vlevo abs 6 / Posición final izq abs 6 / Position finale gauche abs 6 / véghelyzet balra abs 6 / Pos finale a sx ass. 6 / Poł. krańc. lewej abs 6 / Конечное положение влево абс. 6 / Ändläge vänster abs 6 / Posição final esq abs 6 / Poziţie de capăt stânga abs 6 / End position left abs 6'; 626 'Bew aktiv rechts sym / Movement active right sym / 右侧运动生效系统 6 / Pohyb akt vpravo sym 6 / Mov act dcha simb 6 / Dépl act droite sym 6 / mozgás aktív jobbra sym 6 / Mov att a dx simm. 6 / Ruch aktyw. lewo sym 6 / Движение активно вправо симв. 6 / Rörelse aktiv höger sym 6 / Movmt atv dir sym 6 / Depl. activă dreapta sim 6 / Movmt act right sym 6'; 627 'Bew aktiv rechts abs / Movement active right abs / 右侧运动生效绝对 6 / Pohyb akt vpravo abs 6 / Mov act dcha abs 6 / Dépl act droite abs 6 / mozgás aktív jobbra abs 6 / Mov att a dx ass. 6 / Ruch aktyw. prawo 6 / Движение активно вправо абс. 6 / Rörelse aktiv höger abs 6 / Movmt atv direito abs 6 / Depl. activă dreapta abs 6 / Movmt act right abs 6'; 628 'Endlage rechts sym / End position right sym / 右侧最终位置系统 6 / Koncová poloha vpravo sym 6 / Posición final dcha simb 6 / Position finale droite sym 6 / véghelyzet jobbra sym 6 / Pos finale a dx simm. 6 / Poł. krańc. prawej sym 6 / Конечное положение вправо симв. 6 / Ändläge höger sym 6 / Posição final dir sym 6 / Poziţie de capăt dreapta sim 6 / End position right sym 6'; 629 'Endlage rechts abs / End position right abs / 右侧最终位置绝对 6 / Koncová poloha vpravo abs 6 / Posición final derecha abs 6 / Position finale droite abs 6 / véghelyzet jobbra absz 6 / Pos finale a dx ass. 6 / Położenie krańcowe prawe abs 6 / Конечное положение вправо abs 6 / Ändläge höger abs 6 / Posição final direita abs 6 / Poziţie de capăt dreapta abs 6 / End position right abs 6'; 630 'Funktion sym / Function sym / 功能系统 6 / Funkce sym 6 / Función simb 6 / Fonction sym 6 / sym 6 funkció / Funzione simm. 6 / Funkcja sym 6 / Функция симв. 6 / Funktion sym 6 / Função sym 6 / Funcţie sim 6 / Function sym 6'; 631 'Funktion abs / Function abs / 功能绝对 6 / Funkce abs 6 / Función abs 6 / Fonction abs 6 / abs 6 funkció / Funzione ass. 6 / Funkcja abs 6 / Функция абс. 6 / Funktion abs 6 / Função abs 6 / Funcţie abs 6 / Function abs 6'; 632 'Bew aktiv links sym / Movement active left sym / 左侧运动生效系统 6 / Pohyb akt vlevo sym 6 / Mov act izq simb 6 / Dépl act gauche sym 6 / mozgás aktív balra sym 6 / Mov att a sx simm. 6 / Ruch aktyw. lewo sym 6 / Движение активно влево симв. 6 / Rörelse aktiv vänster sym 6 / Movmt atv esq sym 6 / Depl. activă stânga sim 6 / Movmt act left sym 6'; 633 'Bew aktiv links abs / Movement active left abs / 左侧运动生效绝对 6 / Pohyb akt vlevo abs 6 / Mov act izq abs 6 / Dépl act gauche abs 6 / mozgás aktív balra abs 6 / Mov att a sx ass. 6 / Ruch aktyw. lewo abs 6 / Движение активно влево абс. 6 / Rörelse aktiv vänster abs 6 / Movmt atv esq abs 6 / Depl. activă stânga abs 6 / Movmt act left abs 6'; 634 'Endlage links sym / End position left sym / 左侧最终位置系统 6 / Koncová poloha vlevo sym 6 / Posición final izq simb 6 / Position finale gauche sym 6 / véghelyzet balra sym 6 / Pos finale a sx simm. 6 / Poł. krańc. lewej sym 6 / Конечное положение влево сим. 6 / Ändläge vänster sym 6 / Posição final esq sym 6 / Poziţie de capăt stânga sim 6 / End position left sym 6'; 635 'Endlage links abs / End position left abs / 左侧最终位置绝对 6 / Koncová poloha vlevo abs 6 / Posición final izq abs 6 / Position finale gauche abs 6 / véghelyzet balra abs 6 / Pos finale a sx ass. 6 / Poł. krańc. lewej abs 6 / Конечное положение влево абс. 6 / Ändläge vänster abs 6 / Posição final esq abs 6 / Poziţie de capăt stânga abs 6 / End position left abs 6'; 636 'Bew aktiv rechts sym / Movement active right sym / 右侧运动生效系统 6 / Pohyb akt vpravo sym 6 / Mov act dcha simb 6 / Dépl act droite sym 6 / mozgás aktív jobbra sym 6 / Mov att a dx simm. 6 / Ruch aktyw. lewo sym 6 / Движение активно вправо симв. 6 / Rörelse aktiv höger sym 6 / Movmt atv dir sym 6 / Depl. activă dreapta sim 6 / Movmt act right sym 6'; 637 'Bew aktiv rechts abs / Movement active right abs / 右侧运动生效绝对 6 / Pohyb akt vpravo abs 6 / Mov act dcha abs 6 / Dépl act droite abs 6 / mozgás aktív jobbra abs 6 / Mov att a dx ass. 6 / Ruch aktyw. prawo 6 / Движение активно вправо абс. 6 / Rörelse aktiv höger abs 6 / Movmt atv direito abs 6 / Depl. activă dreapta abs 6 / Movmt act right abs 6'; 638 'Endlage rechts sym / End position right sym / 右侧最终位置系统 6 / Koncová poloha vpravo sym 6 / Posición final dcha simb 6 / Position finale droite sym 6 / véghelyzet jobbra sym 6 / Pos finale a dx simm. 6 / Poł. krańc. prawej sym 6 / Конечное положение вправо симв. 6 / Ändläge höger sym 6 / Posição final dir sym 6 / Poziţie de capăt dreapta sim 6 / End position right sym 6'; 639 'Endlage rechts abs / End position right abs / 右侧最终位置绝对 6 / Koncová poloha vpravo abs 6 / Posición final derecha abs 6 / Position finale droite abs 6 / véghelyzet jobbra absz 6 / Pos finale a dx ass. 6 / Położenie krańcowe prawe abs 6 / Конечное положение вправо abs 6 / Ändläge höger abs 6 / Posição final direita abs 6 / Poziţie de capăt dreapta abs 6 / End position right abs 6'

text list "Overview": 1 'FG 1'; 2 'FG 2'; 3 'FG 3'; 4 'FG 4'; 5 'FG 5'; 10 'FG Transport'; 0 'FG x'

text list "Header_Line_2": 0 ''; 1 ''

text list "StationState": 0 'Bearbeitung / Processing'; 1 'Störung / Fault'; 2 'Nicht benötigt / Not required'; 3 'Nicht in Produktion / Not in production'; 4 'Wartet auf Bediener / Waiting for operator'; 5 'Ausgabe blockiert / Output blocked'; 6 'Wartet auf Eingabe / Waiting for infeed'

Template "Vorlage_1" 800x420
   Button "Beenden" at 720,360 size 78x58; TextOff 'Beenden / Exit'; PictureOff "ExitRuntime_TP700_Comfort_TR"; PictureOn "ExitRuntime_TP700_Comfort_TR"
      on Release: StopRuntime(0)
   Button "Template_Button" at 640,360 size 78x58; TextOff 'Meldungen / Messages'; PictureOff "meldungen_48"
      on Click: function_ef3f5d25("Meldefenster_Anstehend", -1)
   Button "Template_Button_1" at 560,360 size 78x58; TextOff 'Text'
   Button "Template_Button_2" at 480,360 size 78x58; TextOff 'Text'
   Button "Template_Button_3" at 400,360 size 78x58; TextOff 'Text'
   Button "Template_Button_4" at 321,360 size 78x58; TextOff 'Text'
   Button "Template_Button_5" at 241,360 size 78x58; TextOff 'Taktzeiten / Cycle times'; PictureOff "taktzeiten_48"
      on Release: ActivateScreen("101_Taktzeiten", 0)
   Button "Template_Button_6" at 161,360 size 78x58; TextOff 'Übersicht / Overview'; PictureOff "uebersicht_48"
      on Release: ActivateScreen("2_Übersicht", 0)
   Button "Template_Button_7" at 81,360 size 78x58; TextOff 'zurück / back'; PictureOff "zurueck_48"
      on Click: function_efd93a16()
   Button "Startbild" at 1,360 size 78x58; TextOff 'Startbild / Start screen'; PictureOff "NavigateHome_TP700_Comfort_TR"; PictureOn "NavigateHome_TP700_Comfort_TR"
      on Release: ActivateScreen("1_Grundbild", 0)
   AlarmView "Meldeanzeige_Nichtquittiert" at 0,0 size 800x20

screen "1_Grundbild" 800x420, template "Vorlage_1"
   on GenerateScreen: SetTag("Header_Line_1", 1)
   Button "HmiScreenItemData" at 36,60 size 159x47; TextOff 'Automatik / Automatic'; PictureOff "Navigates to Automatik for TP700 Comfort 17.0.0.0"; PictureOn "Navigates to Automatik for TP700 Comfort 17.0.0.0"
      on Release: ActivateScreen("100_Automatik", 0)
   Button "HmiScreenItemData_1" at 36,119 size 159x47; TextOff 'Einrichten / Setup'; PictureOff "Navigates to Einrichten for TP700 Comfort 17.0.0.0"; PictureOn "Navigates to Einrichten for TP700 Comfort 17.0.0.0"
      on Release: ActivateScreen("10_Einrichten", 0)
   Button "HmiScreenItemData_3" at 36,178 size 159x47; TextOff 'Systembilder / System screens'; PictureOff "Navigates to Systembilder for TP700 Comfort 17.0.0.0"; PictureOn "Navigates to Systembilder for TP700 Comfort 17.0.0.0"
      on Release: ActivateScreen("1000_Systembilder", 0)

screen "100_Automatik" 800x420, template "Vorlage_1"
   on GenerateScreen: SetTag("Header_Line_1", 100)
   TextField "Textfeld_1" at 11,34 size 365x42; Text 'Maschine leerfahren / Empty machine'
   Switch "Schalter_1" at 376,34 size 83x42; CaptionText 'Umschalten'; TextOff 'Aus / Off'; TextOn 'Ein / On'
      ProcessValue <- "MachineGlobals_emptying"
      Appearance <- "MachineGlobals_emptying"
   TextField "Textfeld_2" at 11,76 size 365x42; Text 'FG05 leerfahren / Empty FG05'
   Switch "Schalter_2" at 376,76 size 83x42; CaptionText 'Umschalten'; TextOff 'Aus / Off'; TextOn 'Ein / On'
      ProcessValue <- "FG05Globals_emptying"
      Appearance <- "FG05Globals_emptying"
   TextField "Textfeld_3" at 11,118 size 365x42; Text 'FG01 Laser einschalten / FG01 Switch on laser'
   Switch "Schalter_3" at 376,118 size 83x42; CaptionText 'Umschalten'; TextOff 'Aus / Off'; TextOn 'Ein / On'
      ProcessValue <- "FG01Globals_laserOn"
      Appearance <- "FG01Globals_laserOn"

screen "10_Einrichten" 800x420, template "Vorlage_1"
   on GenerateScreen: SetTag("Header_Line_1", 10)
   Button "HmiScreenItemData_1" at 35,41 size 159x47; TextOff 'FG 1 / Einrichtfunktionen'; TextOn 'Einrichtfunktionen'; PictureOff "Navigates to Einrichtfunktionen for TP700 Comfort 17.0.0.0"; PictureOn "Navigates to Einrichtfunktionen for TP700 Comfort 17.0.0.0"
      on Release: ActivateScreen("12_Einrichtfunktionen", 0); SetTag("HmiManualMovement_selection_station", 1)
      Visibility <- "xExists"
   Button "HmiScreenItemData_2" at 35,100 size 159x47; TextOff 'FG 2 / Einrichtfunktionen'; TextOn 'Einrichtfunktionen'; PictureOff "Navigates to Einrichtfunktionen for TP700 Comfort 17.0.0.0"; PictureOn "Navigates to Einrichtfunktionen for TP700 Comfort 17.0.0.0"
      on Release: ActivateScreen("12_Einrichtfunktionen", 0); SetTag("HmiManualMovement_selection_station", 2)
      Visibility <- "xExists"
   Button "HmiScreenItemData_3" at 35,160 size 159x47; TextOff 'FG 3 / Einrichtfunktionen'; TextOn 'Einrichtfunktionen'; PictureOff "Navigates to Einrichtfunktionen for TP700 Comfort 17.0.0.0"; PictureOn "Navigates to Einrichtfunktionen for TP700 Comfort 17.0.0.0"
      on Release: ActivateScreen("12_Einrichtfunktionen", 0); SetTag("HmiManualMovement_selection_station", 3)
      Visibility <- "xExists"
   Button "HmiScreenItemData_4" at 35,223 size 159x47; TextOff 'FG 4 / Einrichtfunktionen'; TextOn 'Einrichtfunktionen'; PictureOff "Navigates to Einrichtfunktionen for TP700 Comfort 17.0.0.0"; PictureOn "Navigates to Einrichtfunktionen for TP700 Comfort 17.0.0.0"
      on Release: ActivateScreen("12_Einrichtfunktionen", 0); SetTag("HmiManualMovement_selection_station", 4)
      Visibility <- "xExists"
   Button "HmiScreenItemData_5" at 35,282 size 159x47; TextOff 'FG 5 / Einrichtfunktionen'; TextOn 'Einrichtfunktionen'; PictureOff "Navigates to Einrichtfunktionen for TP700 Comfort 17.0.0.0"; PictureOn "Navigates to Einrichtfunktionen for TP700 Comfort 17.0.0.0"
      on Release: ActivateScreen("12_Einrichtfunktionen", 0); SetTag("HmiManualMovement_selection_station", 5)
      Visibility <- "xExists"
   Button "HmiScreenItemData_6" at 232,282 size 159x47; TextOff 'FG Transport / Einrichtfunktionen'; TextOn 'Einrichtfunktionen'; PictureOff "Navigates to Einrichtfunktionen for TP700 Comfort 17.0.0.0"; PictureOn "Navigates to Einrichtfunktionen for TP700 Comfort 17.0.0.0"
      on Release: ActivateScreen("12_Einrichtfunktionen", 0); SetTag("HmiManualMovement_selection_station", 10)
      Visibility <- "xExists"
   Button "HmiScreenItemData_7" at 232,41 size 159x47; TextOff 'FG 6 / Einrichtfunktionen'; TextOn 'Einrichtfunktionen'; PictureOff "Navigates to Einrichtfunktionen for TP700 Comfort 17.0.0.0"; PictureOn "Navigates to Einrichtfunktionen for TP700 Comfort 17.0.0.0"
      on Release: ActivateScreen("12_Einrichtfunktionen", 0); SetTag("HmiManualMovement_selection_station", 1)
      Visibility <- "xExists"
   Button "HmiScreenItemData_8" at 232,100 size 159x47; TextOff 'FG 7 / Einrichtfunktionen'; TextOn 'Einrichtfunktionen'; PictureOff "Navigates to Einrichtfunktionen for TP700 Comfort 17.0.0.0"; PictureOn "Navigates to Einrichtfunktionen for TP700 Comfort 17.0.0.0"
      on Release: ActivateScreen("12_Einrichtfunktionen", 0); SetTag("HmiManualMovement_selection_station", 1)
      Visibility <- "xExists"
   Button "HmiScreenItemData_9" at 232,159 size 159x47; TextOff 'FG 8 / Einrichtfunktionen'; TextOn 'Einrichtfunktionen'; PictureOff "Navigates to Einrichtfunktionen for TP700 Comfort 17.0.0.0"; PictureOn "Navigates to Einrichtfunktionen for TP700 Comfort 17.0.0.0"
      on Release: ActivateScreen("12_Einrichtfunktionen", 0); SetTag("HmiManualMovement_selection_station", 1)
      Visibility <- "xExists"
   Button "HmiScreenItemData_10" at 232,218 size 159x47; TextOff 'FG 9 / Einrichtfunktionen'; TextOn 'Einrichtfunktionen'; PictureOff "Navigates to Einrichtfunktionen for TP700 Comfort 17.0.0.0"; PictureOn "Navigates to Einrichtfunktionen for TP700 Comfort 17.0.0.0"
      on Release: ActivateScreen("12_Einrichtfunktionen", 0); SetTag("HmiManualMovement_selection_station", 1)
      Visibility <- "xExists"

screen "12_Einrichtfunktionen" 800x420, template "Vorlage_1"
   on GenerateScreen: SetTag("Header_Line_1", 12); SetTag("Header_Line_2", 1)
   on ClearScreen: SetTag("HmiManualMovement_selection_station", 0); SetTag("Header_Line_2", 0)
   Rectangle "recExecuteLeft1" at 0,22 size 285x72
      Visibility <- "showRecLeft"
   Rectangle "recRuntime1" at 287,22 size 226x72
      Visibility <- "showName"
   Rectangle "recExecuteRight1" at 515,22 size 285x72
      Visibility <- "showRecRight"
   Rectangle "recConfirmExecuteLeft1" at 60,26 size 29x29
      Appearance <- "workAct"
      Visibility <- "isExecutableLeft"
   Rectangle "recFinalPositionLeft1" at 60,61 size 29x29
      Appearance <- "inWorkPos"
      Visibility <- "hasEndPositionLeft"
   Polygon "polExecutabilityLeft1" at 2,30 size 51x55
      Appearance <- "workIsInterlocked"
      Visibility <- "isExecutableLeft"
   SymbolicIOField "seaConfirmExecuteLeft1" at 92,26 size 193x29; TextOn '1'; TextOff '0'; TextList "Setup"
      ProcessValue <- "textlistFunctionExecuteLeft"
      Visibility <- "isExecutableLeft"
   SymbolicIOField "seaFinalPositionLeft1" at 92,61 size 193x29; TextOn '1'; TextOff '0'; TextList "Setup"
      ProcessValue <- "textlistFunctionFinalPosLeft"
      Visibility <- "hasEndPositionLeft"
   Rectangle "recFinalPositionRight1" at 711,61 size 29x29
      Appearance <- "inHomePos"
      Visibility <- "hasEndPositionRight"
   Polygon "polExecutabilityRight1" at 747,30 size 51x55
      Appearance <- "homeIsInterlocked"
      Visibility <- "isExecutableRight"
   SymbolicIOField "seaFunction1" at 287,26 size 226x29; TextOn '1'; TextOff '0'; TextList "Setup"
      ProcessValue <- "textlistFunctionName"
      Visibility <- "showName"
   SymbolicIOField "seaConfirmExecuteRight1" at 515,26 size 193x29; TextOn '1'; TextOff '0'; TextList "Setup"
      ProcessValue <- "textlistFunctionExecuteRight"
      Visibility <- "isExecutableRight"
   SymbolicIOField "seaFinalPositionRight1" at 515,61 size 193x29; TextOn '1'; TextOff '0'; TextList "Setup"
      ProcessValue <- "textlistFunctionFinalPosRight"
      Visibility <- "hasEndPositionRight"
   IOField "eaPosition1" at 287,61 size 226x29; FormatPattern s999999999.999
      ProcessValue <- "value"
      Visibility <- "showValue"
   Rectangle "recConfirmExecuteRight1" at 711,26 size 29x29
      Appearance <- "homeAct"
      Visibility <- "isExecutableRight"
   Button "btnRight1" at 515,22 size 285x72; TextOn 'Texto / Texte / Testo / 文本 / Text / Szöv / Текст / Tekst'; TextOff 'Texto / Texte / Testo / 文本 / Text / Szöv / Текст / Tekst'
      on Release: SetTag("moveHomePos", 0)
      on Press: SetTag("moveHomePos", 1)
      ObjectEnable <- "isExecutableRight"
   Button "btnLeft1" at 0,22 size 285x72; TextOn 'Texto / Texte / Testo / 文本 / Text / Szöv / Текст / Tekst'; TextOff 'Texto / Texte / Testo / 文本 / Text / Szöv / Текст / Tekst'
      on Release: SetTag("moveWorkPos", 0)
      on Press: SetTag("moveWorkPos", 1)
      ObjectEnable <- "isExecutableLeft"
   TextField "txtPage" at 524,326 size 120x29; Text 'Seite / Página / Page / Pagina / 页 / Stránka / Oldal / Страница / stron / Sida / Pagină'
   IOField "eaActualPage" at 654,326 size 41x29; FormatPattern 999
      ProcessValue <- "HmiManualMovement_selection_page"
   TextField "txtOf" at 696,326 size 56x29; Text 'von / de / di / 之 / of / od / tól / из / z / av / din'
   IOField "eaNumberOfPages" at 753,326 size 41x29; FormatPattern 999
      ProcessValue <- "HmiManualMovement_selection_ofMaxPages"
   Group "Function 1" at 0,22 size 800x72; TextList "Setup"
   Group "Function 2" at 0,96 size 800x72; TextList "Setup"
   Group "Function 3" at 0,170 size 800x72; TextList "Setup"
   Group "Function 4" at 0,244 size 800x72; TextList "Setup"
   Button "Template_Button" at 640,360 size 78x58; TextOff 'Seite + Page +'; PictureOff "seite_vor_48"
      on Press: SetBit("HmiManualMovement_selection_nextPage")
   Button "Template_Button_1" at 560,360 size 78x58; TextOff 'Seite - Page -'; PictureOff "seite_zurueck_48"
      on Press: SetBit("HmiManualMovement_selection_previousPage")
   Button "Template_Button_2" at 480,360 size 78x58; TextOff 'Symbol Absolut Symbolic Absolute'; PictureOff "symbol_absolut_48"
      on Press: InvertBit("HmiManualMovement_selection_showSymbols")
   Rectangle "recExecuteLeft1_1" at 0,96 size 285x72
      Visibility <- "showRecLeft"
   Rectangle "recRuntime1_1" at 287,96 size 226x72
      Visibility <- "showName"
   Rectangle "recExecuteRight1_1" at 515,96 size 285x72
      Visibility <- "showRecRight"
   Rectangle "recConfirmExecuteLeft1_1" at 60,100 size 29x29
      Appearance <- "workAct"
      Visibility <- "isExecutableLeft"
   Rectangle "recFinalPositionLeft1_1" at 60,135 size 29x29
      Appearance <- "inWorkPos"
      Visibility <- "hasEndPositionLeft"
   Polygon "polExecutabilityLeft1_1" at 2,104 size 51x55
      Appearance <- "workIsInterlocked"
      Visibility <- "isExecutableLeft"
   SymbolicIOField "seaConfirmExecuteLeft1_1" at 92,100 size 193x29; TextOn '1'; TextOff '0'; TextList "Setup"
      ProcessValue <- "textlistFunctionExecuteLeft"
      Visibility <- "isExecutableLeft"
   SymbolicIOField "seaFinalPositionLeft1_1" at 92,135 size 193x29; TextOn '1'; TextOff '0'; TextList "Setup"
      ProcessValue <- "textlistFunctionFinalPosLeft"
      Visibility <- "hasEndPositionLeft"
   Rectangle "recFinalPositionRight1_1" at 711,135 size 29x29
      Appearance <- "inHomePos"
      Visibility <- "hasEndPositionRight"
   Polygon "polExecutabilityRight1_1" at 747,104 size 51x55
      Appearance <- "homeIsInterlocked"
      Visibility <- "isExecutableRight"
   SymbolicIOField "seaFunction1_1" at 287,100 size 226x29; TextOn '1'; TextOff '0'; TextList "Setup"
      ProcessValue <- "textlistFunctionName"
      Visibility <- "showName"
   SymbolicIOField "seaConfirmExecuteRight1_1" at 515,100 size 193x29; TextOn '1'; TextOff '0'; TextList "Setup"
      ProcessValue <- "textlistFunctionExecuteRight"
      Visibility <- "isExecutableRight"
   SymbolicIOField "seaFinalPositionRight1_1" at 515,135 size 193x29; TextOn '1'; TextOff '0'; TextList "Setup"
      ProcessValue <- "textlistFunctionFinalPosRight"
      Visibility <- "hasEndPositionRight"
   IOField "eaPosition1_1" at 287,135 size 226x29; FormatPattern s999999999.999
      ProcessValue <- "value"
      Visibility <- "showValue"
   Rectangle "recConfirmExecuteRight1_1" at 711,100 size 29x29
      Appearance <- "homeAct"
      Visibility <- "isExecutableRight"
   Button "btnRight1_1" at 515,96 size 285x72; TextOn 'Texto / Texte / Testo / 文本 / Text / Szöv / Текст / Tekst'; TextOff 'Texto / Texte / Testo / 文本 / Text / Szöv / Текст / Tekst'
      on Release: SetTag("moveHomePos", 0)
      on Press: SetTag("moveHomePos", 1)
      ObjectEnable <- "isExecutableRight"
   Button "btnLeft1_1" at 0,96 size 285x72; TextOn 'Texto / Texte / Testo / 文本 / Text / Szöv / Текст / Tekst'; TextOff 'Texto / Texte / Testo / 文本 / Text / Szöv / Текст / Tekst'
      on Release: SetTag("moveWorkPos", 0)
      on Press: SetTag("moveWorkPos", 1)
      ObjectEnable <- "isExecutableLeft"
   Rectangle "recExecuteLeft1_2" at 0,170 size 285x72
      Visibility <- "showRecLeft"
   Rectangle "recRuntime1_2" at 287,170 size 226x72
      Visibility <- "showName"
   Rectangle "recExecuteRight1_2" at 515,170 size 285x72
      Visibility <- "showRecRight"
   Rectangle "recConfirmExecuteLeft1_2" at 60,174 size 29x29
      Appearance <- "workAct"
      Visibility <- "isExecutableLeft"
   Rectangle "recFinalPositionLeft1_2" at 60,209 size 29x29
      Appearance <- "inWorkPos"
      Visibility <- "hasEndPositionLeft"
   Polygon "polExecutabilityLeft1_2" at 2,178 size 51x55
      Appearance <- "workIsInterlocked"
      Visibility <- "isExecutableLeft"
   SymbolicIOField "seaConfirmExecuteLeft1_2" at 92,174 size 193x29; TextOn '1'; TextOff '0'; TextList "Setup"
      ProcessValue <- "textlistFunctionExecuteLeft"
      Visibility <- "isExecutableLeft"
   SymbolicIOField "seaFinalPositionLeft1_2" at 92,209 size 193x29; TextOn '1'; TextOff '0'; TextList "Setup"
      ProcessValue <- "textlistFunctionFinalPosLeft"
      Visibility <- "hasEndPositionLeft"
   Rectangle "recFinalPositionRight1_2" at 711,209 size 29x29
      Appearance <- "inHomePos"
      Visibility <- "hasEndPositionRight"
   Polygon "polExecutabilityRight1_2" at 747,178 size 51x55
      Appearance <- "homeIsInterlocked"
      Visibility <- "isExecutableRight"
   SymbolicIOField "seaFunction1_2" at 287,174 size 226x29; TextOn '1'; TextOff '0'; TextList "Setup"
      ProcessValue <- "textlistFunctionName"
      Visibility <- "showName"
   SymbolicIOField "seaConfirmExecuteRight1_2" at 515,174 size 193x29; TextOn '1'; TextOff '0'; TextList "Setup"
      ProcessValue <- "textlistFunctionExecuteRight"
      Visibility <- "isExecutableRight"
   SymbolicIOField "seaFinalPositionRight1_2" at 515,209 size 193x29; TextOn '1'; TextOff '0'; TextList "Setup"
      ProcessValue <- "textlistFunctionFinalPosRight"
      Visibility <- "hasEndPositionRight"
   IOField "eaPosition1_2" at 287,209 size 226x29; FormatPattern s999999999.999
      ProcessValue <- "value"
      Visibility <- "showValue"
   Rectangle "recConfirmExecuteRight1_2" at 711,174 size 29x29
      Appearance <- "homeAct"
      Visibility <- "isExecutableRight"
   Button "btnRight1_2" at 515,170 size 285x72; TextOn 'Texto / Texte / Testo / 文本 / Text / Szöv / Текст / Tekst'; TextOff 'Texto / Texte / Testo / 文本 / Text / Szöv / Текст / Tekst'
      on Release: SetTag("moveHomePos", 0)
      on Press: SetTag("moveHomePos", 1)
      ObjectEnable <- "isExecutableRight"
   Button "btnLeft1_2" at 0,170 size 285x72; TextOn 'Texto / Texte / Testo / 文本 / Text / Szöv / Текст / Tekst'; TextOff 'Texto / Texte / Testo / 文本 / Text / Szöv / Текст / Tekst'
      on Release: SetTag("moveWorkPos", 0)
      on Press: SetTag("moveWorkPos", 1)
      ObjectEnable <- "isExecutableLeft"
   Rectangle "recExecuteLeft1_3" at 0,244 size 285x72
      Visibility <- "showRecLeft"
   Rectangle "recRuntime1_3" at 287,244 size 226x72
      Visibility <- "showName"
   Rectangle "recExecuteRight1_3" at 515,244 size 285x72
      Visibility <- "showRecRight"
   Rectangle "recConfirmExecuteLeft1_3" at 60,248 size 29x29
      Appearance <- "workAct"
      Visibility <- "isExecutableLeft"
   Rectangle "recFinalPositionLeft1_3" at 60,283 size 29x29
      Appearance <- "inWorkPos"
      Visibility <- "hasEndPositionLeft"
   Polygon "polExecutabilityLeft1_3" at 2,252 size 51x55
      Appearance <- "workIsInterlocked"
      Visibility <- "isExecutableLeft"
   SymbolicIOField "seaConfirmExecuteLeft1_3" at 92,248 size 193x29; TextOn '1'; TextOff '0'; TextList "Setup"
      ProcessValue <- "textlistFunctionExecuteLeft"
      Visibility <- "isExecutableLeft"
   SymbolicIOField "seaFinalPositionLeft1_3" at 92,283 size 193x29; TextOn '1'; TextOff '0'; TextList "Setup"
      ProcessValue <- "textlistFunctionFinalPosLeft"
      Visibility <- "hasEndPositionLeft"
   Rectangle "recFinalPositionRight1_3" at 711,283 size 29x29
      Appearance <- "inHomePos"
      Visibility <- "hasEndPositionRight"
   Polygon "polExecutabilityRight1_3" at 747,252 size 51x55
      Appearance <- "homeIsInterlocked"
      Visibility <- "isExecutableRight"
   SymbolicIOField "seaFunction1_3" at 287,248 size 226x29; TextOn '1'; TextOff '0'; TextList "Setup"
      ProcessValue <- "textlistFunctionName"
      Visibility <- "showName"
   SymbolicIOField "seaConfirmExecuteRight1_3" at 515,248 size 193x29; TextOn '1'; TextOff '0'; TextList "Setup"
      ProcessValue <- "textlistFunctionExecuteRight"
      Visibility <- "isExecutableRight"
   SymbolicIOField "seaFinalPositionRight1_3" at 515,283 size 193x29; TextOn '1'; TextOff '0'; TextList "Setup"
      ProcessValue <- "textlistFunctionFinalPosRight"
      Visibility <- "hasEndPositionRight"
   IOField "eaPosition1_3" at 287,283 size 226x29; FormatPattern s999999999.999
      ProcessValue <- "value"
      Visibility <- "showValue"
   Rectangle "recConfirmExecuteRight1_3" at 711,248 size 29x29
      Appearance <- "homeAct"
      Visibility <- "isExecutableRight"
   Button "btnRight1_3" at 515,244 size 285x72; TextOn 'Texto / Texte / Testo / 文本 / Text / Szöv / Текст / Tekst'; TextOff 'Texto / Texte / Testo / 文本 / Text / Szöv / Текст / Tekst'
      on Release: SetTag("moveHomePos", 0)
      on Press: SetTag("moveHomePos", 1)
      ObjectEnable <- "isExecutableRight"
   Button "btnLeft1_3" at 0,244 size 285x72; TextOn 'Texto / Texte / Testo / 文本 / Text / Szöv / Текст / Tekst'; TextOff 'Texto / Texte / Testo / 文本 / Text / Szöv / Текст / Tekst'
      on Release: SetTag("moveWorkPos", 0)
      on Press: SetTag("moveWorkPos", 1)
      ObjectEnable <- "isExecutableLeft"

screen "1000_Systembilder" 800x420, template "Vorlage_1"
   on GenerateScreen: SetTag("Header_Line_1", 1000)
   Button "Zurück" at 1,25 size 159x47; TextOff 'Zurück / Back'
      on Release: ActivateScreen("1_Grundbild", 0)
   Button "HmiScreenItemData" at 36,119 size 159x47; TextOff 'SIMATIC PLC Systemdiagnose SIMATIC PLC system diagnostics SIMATIC PLC system diagnos...'; PictureOff "Navigates to SIMATIC PLC Systemdiagnose for TP700 Comfort 17.0.0.0"; PictureOn "Navigates to SIMATIC PLC Systemdiagnose for TP700 Comfort 17.0.0.0"
      on Release: ActivateScreen("1001_SIMATIC PLC Systemdiagnose", 0)
   Button "HmiScreenItemData_1" at 36,178 size 159x47; TextOff 'Projektinformationen Project information Project information'; PictureOff "Navigates to Projektinformationen for TP700 Comfort 17.0.0.0"; PictureOn "Navigates to Projektinformationen for TP700 Comfort 17.0.0.0"
      on Release: ActivateScreen("1002_Projektinformationen", 0)
   Button "HmiScreenItemData_2" at 36,237 size 159x47; TextOff 'Systemeinstellungen / System settings'; PictureOff "Navigates to Systemeinstellungen for TP700 Comfort 17.0.0.0"; PictureOn "Navigates to Systemeinstellungen for TP700 Comfort 17.0.0.0"
      on Release: ActivateScreen("1003_Systemeinstellungen", 0)
   Button "HmiScreenItemData_3" at 36,296 size 159x47; TextOff 'Benutzerverwaltung User administration User administration'; PictureOff "Navigates to Benutzerverwaltung for TP700 Comfort 17.0.0.0"; PictureOn "Navigates to Benutzerverwaltung for TP700 Comfort 17.0.0.0"
      on Release: ActivateScreen("1004_Benutzerverwaltung", 0)
   Button "HmiScreenItemData_4" at 207,119 size 159x47; TextOff 'Systeminformationen System information System information'; PictureOff "Navigates to Systeminformationen for TP700 Comfort 17.0.0.0"; PictureOn "Navigates to Systeminformationen for TP700 Comfort 17.0.0.0"
      on Release: ActivateScreen("1005_Systeminformationen", 0)
   Button "HmiScreenItemData_5" at 207,178 size 159x47; TextOff 'Verschiedene Aufgaben Different jobs'; PictureOff "Navigates to Verschiedene Aufgaben for TP700 Comfort 17.0.0.0"; PictureOn "Navigates to Verschiedene Aufgaben for TP700 Comfort 17.0.0.0"
      on Release: ActivateScreen("1006_Verschiedene Aufgaben", 0)
   Button "HmiScreenItemData_6" at 207,237 size 159x47; TextOff 'Verschiedene Aufgaben Different jobs'; PictureOff "Navigates to Verschiedene Aufgaben for TP700 Comfort 17.0.0.0"; PictureOn "Navigates to Verschiedene Aufgaben for TP700 Comfort 17.0.0.0"
      on Release: ActivateScreen("1006_Verschiedene Aufgaben", 0)

screen "1001_SIMATIC PLC Systemdiagnose" 800x420, template "Vorlage_1"
   on GenerateScreen: SetTag("Header_Line_1", 1001)
   SysDiagControl "HmiScreenItemData" at 1,73 size 796x280
   Button "Zurück" at 1,25 size 159x47; TextOff 'Zurück / Back'
      on Release: ActivateScreen("1000_Systembilder", 0)

screen "1002_Projektinformationen" 800x420, template "Vorlage_1"
   on GenerateScreen: SetTag("Header_Line_1", 1002)
   TextField "HmiScreenItemData" at 35,75 size 171x28; Text 'Projektname: / Project name:'
   TextField "HmiScreenItemData_1" at 241,75 size 524x28; Text 'DT_PSA_OPCV / Testprojekt_RV'
   TextField "HmiScreenItemData_2" at 35,105 size 171x28; Text 'Erstellt: / Created on:'
   TextField "HmiScreenItemData_3" at 241,105 size 524x28; Text '26.09.2026 14:49:17 / 26/09/2026 14:49:17 / 09.09.2024 14:49:17'
   TextField "HmiScreenItemData_4" at 35,135 size 171x28; Text 'Autor: / Author:'
   TextField "HmiScreenItemData_5" at 241,135 size 524x28; Text 'Andreas Fast Automation / AFA'
   TextField "HmiScreenItemData_6" at 35,165 size 171x28; Text 'Beschreibung: / Description:'
   TextField "HmiScreenItemData_7" at 241,165 size 524x28; Text '(nicht konfiguriert) / (not configured)'
   Button "Zurück" at 1,25 size 159x47; TextOff 'Zurück / Back'
      on Release: ActivateScreen("1000_Systembilder", 0)

screen "1003_Systemeinstellungen" 800x420, template "Vorlage_1"
   on GenerateScreen: SetTag("Header_Line_1", 1003)
   Button "Bildschirm kalibrieren" at 36,119 size 159x47; TextOff 'Bildschirm kalibrieren / Calibrate screen'
      on Release: function_bc3e350c()
   Button "Putzbild" at 36,178 size 159x47; TextOff 'Putzbild / Clean screen'
      on Release: function_be740847(30)
   Button "Zurück" at 1,25 size 159x47; TextOff 'Zurück / Back'
      on Release: ActivateScreen("1000_Systembilder", 0)

screen "1004_Benutzerverwaltung" 800x420, template "Vorlage_1"
   on GenerateScreen: SetTag("Header_Line_1", 1004)
   UserView "HmiScreenItemData" at 1,73 size 796x280
   Button "Zurück" at 1,25 size 159x47; TextOff 'Zurück / Back'
      on Release: ActivateScreen("1000_Systembilder", 0)

screen "1005_Systeminformationen" 800x420, template "Vorlage_1"
   on GenerateScreen: SetTag("Header_Line_1", 1005)
   TextField "HmiScreenItemData" at 35,75 size 171x28; Text 'Bediengerätetyp: / HMI device type:'
   TextField "HmiScreenItemData_1" at 241,75 size 524x28; Text 'TP700 Comfort 17.0.0.0'
   TextField "HmiScreenItemData_2" at 35,105 size 171x28; Text 'Version:'
   TextField "HmiScreenItemData_3" at 35,135 size 171x28; Text 'Verbindung: / Connection:'
   TextField "HmiScreenItemData_4" at 241,135 size 524x28; Text 'ETHERNET'
   TextField "HmiScreenItemData_5" at 35,165 size 171x28; Text 'Steuerung: / PLC:'
   TextField "HmiScreenItemData_6" at 241,165 size 524x28; Text 'SIMATIC S7 1500'
   Button "Version anzeigen" at 241,105 size 524x28; TextOff 'Version anzeigen / Display version'
      on Release: function_febcb963(-1)
   Button "Zurück" at 1,25 size 159x47; TextOff 'Zurück / Back'
      on Release: ActivateScreen("1000_Systembilder", 0)

screen "1006_Verschiedene Aufgaben" 800x420, template "Vorlage_1"
   on GenerateScreen: SetTag("Header_Line_1", 1006)
   Button "Online" at 36,119 size 159x47; TextOff 'Online'
      on Release: function_bb44b551(0)
   Button "Offline" at 36,178 size 159x47; TextOff 'Offline'
      on Release: function_bb44b551(1)
   Button "Transfer" at 36,237 size 159x47; TextOff 'Transfer'
      on Release: function_bb44b551(2)
   Button "Sprache umschalten" at 36,296 size 159x47; TextOff 'Sprache umschalten / Toggle language'
      on Release: function_fb9197e8(-1)
   Button "Systemsteuerung" at 207,119 size 159x47; TextOff 'Systemsteuerung / Control Panel'
      on Release: function_f34a74f3()
   Button "Runtime beenden" at 207,178 size 159x47; TextOff 'Runtime beenden / Stop Runtime'
      on Release: StopRuntime(0)
   Button "Zurück" at 1,25 size 159x47; TextOff 'Zurück / Back'
      on Release: ActivateScreen("1000_Systembilder", 0)

screen "2_Übersicht" 800x420, template "Vorlage_1"
   on GenerateScreen: SetTag("Header_Line_1", 2)
   SymbolicIOField "Symbolisches_EA_Feld_Bild" at 47,80 size 365x42; TextOff '0'; TextOn '1'; TextList "Overview"
      ProcessValue <- "Übersicht_Station1"
   GraphicIOField "Vorlage_Grafisches EA-Feld_3" at 499,79 size 42x42; PictureOff "manual_off"; PictureOn "manual_on"
      ProcessValue <- "modeSetup"
   GraphicIOField "Vorlage_Grafisches EA-Feld_5" at 585,79 size 42x42; PictureOff "home_off"; PictureOn "home_on"
      ProcessValue <- "isInHome"
   GraphicIOField "Vorlage_Grafisches EA-Feld_6" at 628,79 size 42x42; PictureOff "homing_off"; PictureOn "homing_on"
      ProcessValue <- "isHoming"
   GraphicIOField "Vorlage_Grafisches EA-Feld_7" at 671,79 size 42x42; PictureOff "autoIsStopping_off"; PictureOn "autoIsStopping_on_blue"
      ProcessValue <- "isInAutoStoping"
   SymbolicIOField "Symbolisches_EA_Feld_Bild_1" at 47,124 size 365x42; TextOff '0'; TextOn '1'; TextList "Overview"
      ProcessValue <- "Übersicht_Station2"
   GraphicIOField "Vorlage_Grafisches EA-Feld_8" at 413,123 size 42x42; PictureOff "auto_off"; PictureOn "auto_on"
      ProcessValue <- "modeAuto"
   GraphicIOField "Vorlage_Grafisches EA-Feld_9" at 456,123 size 42x42; PictureOff "step_off"; PictureOn "step_on"
      ProcessValue <- "modeTap"
   GraphicIOField "Vorlage_Grafisches EA-Feld_10" at 499,123 size 42x42; PictureOff "manual_off"; PictureOn "manual_on"
      ProcessValue <- "modeSetup"
   GraphicIOField "Vorlage_Grafisches EA-Feld_11" at 542,123 size 42x42; PictureOff "cycle_off"; PictureOn "cycle_on"
      ProcessValue <- "releaseCycle"
   GraphicIOField "Vorlage_Grafisches EA-Feld_12" at 585,123 size 42x42; PictureOff "home_off"; PictureOn "home_on"
      ProcessValue <- "isInHome"
   GraphicIOField "Vorlage_Grafisches EA-Feld_13" at 628,123 size 42x42; PictureOff "homing_off"; PictureOn "homing_on"
      ProcessValue <- "isHoming"
   GraphicIOField "Vorlage_Grafisches EA-Feld_14" at 671,123 size 42x42; PictureOff "autoIsStopping_off"; PictureOn "autoIsStopping_on_blue"
      ProcessValue <- "isInAutoStoping"
   SymbolicIOField "Symbolisches_EA_Feld_Bild_2" at 47,168 size 365x42; TextOff '0'; TextOn '1'; TextList "Overview"
      ProcessValue <- "Übersicht_Station3"
   GraphicIOField "Vorlage_Grafisches EA-Feld_15" at 413,167 size 42x42; PictureOff "auto_off"; PictureOn "auto_on"
      ProcessValue <- "modeAuto"
   GraphicIOField "Vorlage_Grafisches EA-Feld_16" at 456,167 size 42x42; PictureOff "step_off"; PictureOn "step_on"
      ProcessValue <- "modeTap"
   GraphicIOField "Vorlage_Grafisches EA-Feld_17" at 499,167 size 42x42; PictureOff "manual_off"; PictureOn "manual_on"
      ProcessValue <- "modeSetup"
   GraphicIOField "Vorlage_Grafisches EA-Feld_18" at 542,167 size 42x42; PictureOff "cycle_off"; PictureOn "cycle_on"
      ProcessValue <- "releaseCycle"
   GraphicIOField "Vorlage_Grafisches EA-Feld_19" at 585,167 size 42x42; PictureOff "home_off"; PictureOn "home_on"
      ProcessValue <- "isInHome"
   GraphicIOField "Vorlage_Grafisches EA-Feld_20" at 628,167 size 42x42; PictureOff "homing_off"; PictureOn "homing_on"
      ProcessValue <- "isHoming"
   GraphicIOField "Vorlage_Grafisches EA-Feld_21" at 671,167 size 42x42; PictureOff "autoIsStopping_off"; PictureOn "autoIsStopping_on_blue"
      ProcessValue <- "isInAutoStoping"
   SymbolicIOField "Symbolisches_EA_Feld_Bild_3" at 47,212 size 365x42; TextOff '0'; TextOn '1'; TextList "Overview"
      ProcessValue <- "Übersicht_Station4"
   GraphicIOField "Vorlage_Grafisches EA-Feld_22" at 413,211 size 42x42; PictureOff "auto_off"; PictureOn "auto_on"
      ProcessValue <- "modeAuto"
   GraphicIOField "Vorlage_Grafisches EA-Feld_23" at 456,211 size 42x42; PictureOff "step_off"; PictureOn "step_on"
      ProcessValue <- "modeTap"
   GraphicIOField "Vorlage_Grafisches EA-Feld_24" at 499,211 size 42x42; PictureOff "manual_off"; PictureOn "manual_on"
      ProcessValue <- "modeSetup"
   GraphicIOField "Vorlage_Grafisches EA-Feld_25" at 542,211 size 42x42; PictureOff "cycle_off"; PictureOn "cycle_on"
      ProcessValue <- "releaseCycle"
   GraphicIOField "Vorlage_Grafisches EA-Feld_26" at 585,211 size 42x42; PictureOff "home_off"; PictureOn "home_on"
      ProcessValue <- "isInHome"
   GraphicIOField "Vorlage_Grafisches EA-Feld_27" at 628,211 size 42x42; PictureOff "homing_off"; PictureOn "homing_on"
      ProcessValue <- "isHoming"
   GraphicIOField "Vorlage_Grafisches EA-Feld_28" at 671,211 size 42x42; PictureOff "autoIsStopping_off"; PictureOn "autoIsStopping_on_blue"
      ProcessValue <- "isInAutoStoping"
   SymbolicIOField "Symbolisches_EA_Feld_Bild_4" at 47,256 size 365x42; TextOff '0'; TextOn '1'; TextList "Overview"
      ProcessValue <- "Übersicht_Station5"
   GraphicIOField "Vorlage_Grafisches EA-Feld_29" at 413,255 size 42x42; PictureOff "auto_off"; PictureOn "auto_on"
      ProcessValue <- "modeAuto"
   GraphicIOField "Vorlage_Grafisches EA-Feld_30" at 456,255 size 42x42; PictureOff "step_off"; PictureOn "step_on"
      ProcessValue <- "modeTap"
   GraphicIOField "Vorlage_Grafisches EA-Feld_31" at 499,255 size 42x42; PictureOff "manual_off"; PictureOn "manual_on"
      ProcessValue <- "modeSetup"
   GraphicIOField "Vorlage_Grafisches EA-Feld_32" at 542,255 size 42x42; PictureOff "cycle_off"; PictureOn "cycle_on"
      ProcessValue <- "releaseCycle"
   GraphicIOField "Vorlage_Grafisches EA-Feld_33" at 585,255 size 42x42; PictureOff "home_off"; PictureOn "home_on"
      ProcessValue <- "isInHome"
   GraphicIOField "Vorlage_Grafisches EA-Feld_34" at 628,255 size 42x42; PictureOff "homing_off"; PictureOn "homing_on"
      ProcessValue <- "isHoming"
   GraphicIOField "Vorlage_Grafisches EA-Feld_35" at 671,255 size 42x42; PictureOff "autoIsStopping_off"; PictureOn "autoIsStopping_on_blue"
      ProcessValue <- "isInAutoStoping"
   SymbolicIOField "Symbolisches_EA_Feld_Bild_5" at 47,300 size 365x42; TextOff '0'; TextOn '1'; TextList "Overview"
      ProcessValue <- "Übersicht_Station10"
   GraphicIOField "Vorlage_Grafisches EA-Feld_36" at 413,299 size 42x42; PictureOff "auto_off"; PictureOn "auto_on"
      ProcessValue <- "modeAuto"
   GraphicIOField "Vorlage_Grafisches EA-Feld_37" at 456,299 size 42x42; PictureOff "step_off"; PictureOn "step_on"
      ProcessValue <- "modeTap"
   GraphicIOField "Vorlage_Grafisches EA-Feld_38" at 499,299 size 42x42; PictureOff "manual_off"; PictureOn "manual_on"
      ProcessValue <- "modeSetup"
   GraphicIOField "Vorlage_Grafisches EA-Feld_39" at 542,299 size 42x42; PictureOff "cycle_off"; PictureOn "cycle_on"
      ProcessValue <- "releaseCycle"
   GraphicIOField "Vorlage_Grafisches EA-Feld_40" at 585,299 size 42x42; PictureOff "home_off"; PictureOn "home_on"
      ProcessValue <- "isInHome"
   GraphicIOField "Vorlage_Grafisches EA-Feld_41" at 628,299 size 42x42; PictureOff "homing_off"; PictureOn "homing_on"
      ProcessValue <- "isHoming"
   GraphicIOField "Vorlage_Grafisches EA-Feld_42" at 671,299 size 42x42; PictureOff "autoIsStopping_off"; PictureOn "autoIsStopping_on_blue"
      ProcessValue <- "isInAutoStoping"
   Switch "Schalter_1" at 414,80 size 42x42; CaptionText 'Umschalten'; TextOff 'AUS'; TextOn 'EIN'; PictureOff "auto_off"; PictureOn "auto_on"
      ProcessValue <- "modeAuto"
   Switch "Schalter_2" at 457,80 size 42x42; CaptionText 'Umschalten'; TextOff 'AUS'; TextOn 'EIN'; PictureOff "step_off"; PictureOn "step_on"
      ProcessValue <- "modeTap"
   Switch "Schalter_3" at 543,80 size 42x42; CaptionText 'Umschalten'; TextOff 'AUS'; TextOn 'EIN'; PictureOff "cycle_off"; PictureOn "cycle_on"
      ProcessValue <- "releaseCycle"
   GraphicIOField "Vorlage_Grafisches EA-Feld_1" at 714,79 size 42x42; PictureOff "fault_off"; PictureOn "fault_on"
      ProcessValue <- "isInError"
   GraphicIOField "Vorlage_Grafisches EA-Feld_2" at 714,123 size 42x42; PictureOff "fault_off"; PictureOn "fault_on"
      ProcessValue <- "isInError"
   GraphicIOField "Vorlage_Grafisches EA-Feld_4" at 714,167 size 42x42; PictureOff "fault_off"; PictureOn "fault_on"
      ProcessValue <- "isInError"
   GraphicIOField "Vorlage_Grafisches EA-Feld_43" at 714,211 size 42x42; PictureOff "fault_off"; PictureOn "fault_on"
      ProcessValue <- "isInError"
   GraphicIOField "Vorlage_Grafisches EA-Feld_44" at 714,255 size 42x42; PictureOff "fault_off"; PictureOn "fault_on"
      ProcessValue <- "isInError"
   GraphicIOField "Vorlage_Grafisches EA-Feld_45" at 714,299 size 42x42; PictureOff "fault_off"; PictureOn "fault_on"
      ProcessValue <- "isInError"
   TextField "Textfeld_1" at 47,28 size 365x42; Text 'Maschine / Machine'
   GraphicIOField "Vorlage_Grafisches EA-Feld_46" at 413,28 size 42x42; PictureOff "manual_on"; PictureOn "auto_on"
      ProcessValue <- "automaticMode"
   Switch "Schalter_4" at 543,28 size 42x42; CaptionText 'Umschalten'; TextOff 'AUS'; TextOn 'EIN'; PictureOff "cycle_off"; PictureOn "cycle_on"
      ProcessValue <- "automaticIsRunning"
   GraphicIOField "Vorlage_Grafisches EA-Feld_47" at 585,27 size 42x42; PictureOff "home_off"; PictureOn "home_on"
      ProcessValue <- "isInHome"
   GraphicIOField "Vorlage_Grafisches EA-Feld_48" at 628,27 size 42x42; PictureOff "homing_off"; PictureOn "homing_on"
      ProcessValue <- "isHoming"
   GraphicIOField "Vorlage_Grafisches EA-Feld_49" at 671,27 size 42x42; PictureOff "autoIsStopping_off"; PictureOn "autoIsStopping_on_blue"
      ProcessValue <- "automaticStops"
   GraphicIOField "Vorlage_Grafisches EA-Feld_50" at 714,27 size 42x42; PictureOff "fault_off"; PictureOn "fault_on"
      ProcessValue <- "isInError"

screen "101_Taktzeiten" 800x420, template "Vorlage_1"
   on GenerateScreen: SetTag("Header_Line_1", 101)
   TextField "Textfeld_1" at 18,52 size 232x42; Text 'FG01'
   IOField "EA-Feld_1" at 413,52 size 81x42; FormatPattern 999.9
      ProcessValue <- "rSetpointSeconds"
   GraphicView "Grafikanzeige_1" at 725,52 size 64x42; Picture "Grafik_3"
      Visibility <- "qiBottleneck"
   TextField "Textfeld_2" at 18,95 size 232x42; Text 'FG02'
   IOField "EA-Feld_3" at 413,95 size 81x42; FormatPattern 999.9
      ProcessValue <- "rSetpointSeconds"
   GraphicView "Grafikanzeige_2" at 725,95 size 64x42; Picture "Grafik_3"
      Visibility <- "qiBottleneck"
   TextField "Textfeld_3" at 18,138 size 232x42; Text 'FG03'
   IOField "EA-Feld_5" at 413,138 size 81x42; FormatPattern 999.9
      ProcessValue <- "rSetpointSeconds"
   GraphicView "Grafikanzeige_3" at 725,138 size 64x42; Picture "Grafik_3"
      Visibility <- "qiBottleneck"
   TextField "Textfeld_4" at 18,181 size 232x42; Text 'FG04'
   IOField "EA-Feld_7" at 413,181 size 81x42; FormatPattern 999.9
      ProcessValue <- "rSetpointSeconds"
   GraphicView "Grafikanzeige_4" at 725,181 size 64x42; Picture "Grafik_3"
      Visibility <- "qiBottleneck"
   TextField "Textfeld_5" at 18,224 size 232x42; Text 'FG05'
   IOField "EA-Feld_9" at 413,224 size 81x42; FormatPattern 999.9
      ProcessValue <- "rSetpointSeconds"
   GraphicView "Grafikanzeige_5" at 725,224 size 64x42; Picture "Grafik_3"
      Visibility <- "qiBottleneck"
   TextField "Textfeld_6" at 714,27 size 84x20; Text 'Engpass / Bottleneck'
      Visibility <- "qiBottleneck"
   Bar "Balken_1" at 496,52 size 228x42; Unit s; MinimumValue 0; MaximumValue 15
      ProcessValue <- "rActiveTimeSeconds"
   TextField "Textfeld_7" at 412,27 size 84x20; Text 'Soll [s] / Target [s]'
   TextField "Textfeld_8" at 496,27 size 229x20; Text 'Letzte Aktivzeit [s] / Last active time [s]'
   Bar "Balken_2" at 496,95 size 228x42; Unit s; MinimumValue 0; MaximumValue 15
      ProcessValue <- "rActiveTimeSeconds"
   Bar "Balken_3" at 496,138 size 228x42; Unit s; MinimumValue 0; MaximumValue 15
      ProcessValue <- "rActiveTimeSeconds"
   Bar "Balken_4" at 496,181 size 228x42; Unit s; MinimumValue 0; MaximumValue 15
      ProcessValue <- "rActiveTimeSeconds"
   Bar "Balken_5" at 496,224 size 228x42; Unit s; MinimumValue 0; MaximumValue 15
      ProcessValue <- "rActiveTimeSeconds"
   TextField "Textfeld_9" at 18,267 size 232x42; Text 'FG Transport'
   IOField "EA-Feld_11" at 413,267 size 81x42; FormatPattern 999.9
      ProcessValue <- "rSetpointSeconds"
   Bar "Balken_6" at 496,267 size 228x42; Unit s; MinimumValue 0; MaximumValue 15
      ProcessValue <- "rActiveTimeSeconds"
   GraphicView "Grafikanzeige_6" at 725,266 size 64x42; Picture "Grafik_3"
      Visibility <- "qiBottleneck"
   SymbolicIOField "Symbolisches EA-Feld_1" at 251,52 size 161x42; TextOff '0'; TextOn '1'; TextList "StationState"
      ProcessValue <- "usiState"
   SymbolicIOField "Symbolisches EA-Feld_2" at 251,95 size 161x42; TextOff '0'; TextOn '1'; TextList "StationState"
      ProcessValue <- "usiState"
   SymbolicIOField "Symbolisches EA-Feld_3" at 251,138 size 161x42; TextOff '0'; TextOn '1'; TextList "StationState"
      ProcessValue <- "usiState"
   SymbolicIOField "Symbolisches EA-Feld_4" at 251,181 size 161x42; TextOff '0'; TextOn '1'; TextList "StationState"
      ProcessValue <- "usiState"
   SymbolicIOField "Symbolisches EA-Feld_5" at 251,224 size 161x42; TextOff '0'; TextOn '1'; TextList "StationState"
      ProcessValue <- "usiState"
   SymbolicIOField "Symbolisches EA-Feld_6" at 251,267 size 161x42; TextOff '0'; TextOn '1'; TextList "StationState"
      ProcessValue <- "usiState"
   TextField "Textfeld_10" at 248,27 size 166x20; Text 'Zustand / State'
   TextField "Textfeld_11" at 17,27 size 220x20; Text 'Station'
   Rectangle "Rechteck_1" at 7,52 size 9x40
      Appearance <- "usiState"
   Rectangle "Rechteck_2" at 7,95 size 9x40
      Appearance <- "usiState"
   Rectangle "Rechteck_3" at 7,138 size 9x40
      Appearance <- "usiState"
   Rectangle "Rechteck_4" at 7,181 size 9x40
      Appearance <- "usiState"
   Rectangle "Rechteck_5" at 7,224 size 9x40
      Appearance <- "usiState"
   Rectangle "Rechteck_6" at 7,267 size 9x40
      Appearance <- "usiState"
*)